# B&R Automation Studio project pneutrunk_plc_interface
Automation Studio 4.9

## Configuration Config1

### Task classes (Cpu.sw)
```
Cyclic#1:
  Client <- Source.UDP.Client.prg
  Narazy <- Source.Narazy.prg [disabled]
  Server <- Source.UDP.Server.prg
  Receiver <- (binary)
  Sender <- (binary)
Cyclic#4:
  Receiver1 <- Source.RS485.Receiver.prg
  Sender1 <- Source.RS485.Sender.prg
  Sensors <- Source.Sensors.prg
DataObjects: Acp10sys
Binaries: FWRules, TCData, udbdef, asfw, User, iomap, sysconf, arconfig, ashwd, Role, ashwac, Acp10map, acp10cfg
Libraries: runtime, AsUDP, asstring, standard, sys_lib, brsystem, dvframe, AsTCP, AsArLog, asieccon, astime, powerlnk, fileio
```

### IoMap.iom - X20CP1684/IoMap.iom
```iecst
VAR_CONFIG
	::modul.tlak2[5] AT %QW."X20CM8281".AnalogOutput01;
	::modul.tlak3[5] AT %QW."X20CM8281a".AnalogOutput01;
	::modul.tlak1[0] AT %QW."X20AO4622".AnalogOutput01;
	::modul.tlak2[0] AT %QW."X20AO4622".AnalogOutput02;
	::modul.tlak3[0] AT %QW."X20AO4622".AnalogOutput03;
	::modul.tlak1[1] AT %QW."X20AO4622".AnalogOutput04;
	::modul.tlak2[1] AT %QW."X20AO4622a".AnalogOutput01;
	::modul.tlak3[1] AT %QW."X20AO4622a".AnalogOutput02;
	::modul.tlak1[2] AT %QW."X20AO4622a".AnalogOutput03;
	::modul.tlak2[2] AT %QW."X20AO4622a".AnalogOutput04;
	::modul.tlak3[2] AT %QW."X20AO4622b".AnalogOutput01;
	::modul.tlak1[3] AT %QW."X20AO4622b".AnalogOutput02;
	::modul.tlak2[3] AT %QW."X20AO4622b".AnalogOutput03;
	::modul.tlak3[3] AT %QW."X20AO4622b".AnalogOutput04;
	::modul.tlak1[4] AT %QW."X20AO4622c".AnalogOutput01;
	::modul.tlak2[4] AT %QW."X20AO4622c".AnalogOutput02;
	::modul.tlak3[4] AT %QW."X20AO4622c".AnalogOutput03;
	::modul.tlak1[5] AT %QW."X20AO4622c".AnalogOutput04;
	::modul.tlakLinear AT %QW."X20CM8281b".AnalogOutput01;
	::modul.tlak2[6] AT %QW."X20AO4622d".AnalogOutput01;
	::modul.tlak3[6] AT %QW."X20AO4622d".AnalogOutput02;
	::modul.tlak1[6] AT %QW."X20AO4622d".AnalogOutput03;
	::buttons.stropCervenaLED AT %QX."X20DO9322".DigitalOutput08;
	::buttons.startLED AT %QX."X20DO9322".DigitalOutput06;
	::buttons.stopLED AT %QX."X20DO9322".DigitalOutput07;
	::buttons.stropBielaLED AT %QX."X20DO9322".DigitalOutput05;
	::buttons.startButton AT %IX."X20DM9324".DigitalInput01;
	::buttons.stop AT %IX."X20DM9324".DigitalInput02;
	::buttons.centralStop AT %IX."X20DM9324".DigitalInput04;
	::buttons.klucik AT %IX."X20DM9324".DigitalInput03;
END_VAR
```

## Logical view

### Global.typ
```iecst
TYPE
	tlacidla : 	STRUCT
		start : BOOL;
		ros : BOOL;
		stopLED : BOOL;
		stop : BOOL;
		startLED : BOOL;
		startButton : BOOL;
		centralStop : BOOL;
		stropBielaLED : BOOL;
		stropCervenaLED : BOOL;
		klucik : BOOL;
	END_STRUCT;
	automatic : 	STRUCT
		y_desired : ARRAY[0..6]OF REAL := [7(0.0)];
		x_desired : ARRAY[0..6]OF REAL := [7(0.0)];
		linear : INT;
		ball_up : BOOL;
		casovac : BOOL;
		effector : BOOL;
		casovac_uchopenie : BOOL;
		ball_piston : BOOL;
		novyCyklus : TIME := T#1s;
		novyCyklusStart : BOOL;
		trajectoryStart2 : BOOL;
		trajectoryTime2 : TIME := T#6s;
		automatic : BOOL;
		holdPosition : BOOL;
		cas : INT;
		box : INT;
		step_color : INT;
		popcorn : BOOL;
		testFarba : INT;
		loptickyVzasobniku : BOOL := TRUE;
		x_desired_previous : ARRAY[0..6]OF INT;
		y_desired_previous : ARRAY[0..6]OF INT;
		I_konstanta : ARRAY[0..6]OF INT;
		levitacia : BOOL;
		desiredPressure2 : ARRAY[0..6]OF INT;
		desiredPressure3 : ARRAY[0..6]OF INT;
		desiredPressure3_previous : ARRAY[0..6]OF INT;
		desiredPressure2_previous : ARRAY[0..6]OF INT;
		desiredPressure1_previous : ARRAY[0..6]OF INT;
		desiredPressureLinear : INT;
		desiredPressure1 : ARRAY[0..6]OF INT;
		step_repeatability : INT;
		handControl : BOOL;
		experiment2 : BOOL;
		experiment3 : BOOL;
		experiment1 : BOOL;
	END_STRUCT;
	packetRS485 : 	STRUCT
		packet : ARRAY[0..9]OF BYTE;
		sendPacketLED : ARRAY[0..5]OF BYTE;
		sendPacketSnimace : ARRAY[0..5]OF BYTE;
		sendPacketFinal : ARRAY[0..5]OF BYTE;
		id : USINT;
	END_STRUCT;
	packetUDP : 	STRUCT
		qLength : INT;
		c : INT;
		q : INT;
		qFull : STRING[80];
		comma : INT;
		qString : ARRAY[0..14]OF STRING[6];
		qDesired : ARRAY[0..14]OF REAL;
		color : INT;
		step : INT;
	END_STRUCT;
	tlaky : 	STRUCT
		tlak3 : USINT;
		tlak2 : USINT;
		tlak1 : USINT;
	END_STRUCT;
	moduly : 	STRUCT
		uhol2 : ARRAY[0..6]OF REAL := [7(0.0)];
		uhol1 : ARRAY[0..6]OF REAL := [7(0.0)];
		koncak : ARRAY[0..6]OF BOOL;
		led : ARRAY[0..6]OF BOOL;
		uholINT2 : INT;
		uholINT1 : INT;
		tlak1 : ARRAY[0..6]OF INT;
		tlak2 : ARRAY[0..6]OF INT;
		tlak3 : ARRAY[0..6]OF INT;
		tlakLinear : INT;
		alpha : ARRAY[0..6]OF REAL; (*uhol ktory posiela PLC do PC po odpocitani odchylky naklonenia realneho robota*)
		beta : ARRAY[0..6]OF REAL; (*uhol ktory posiela PLC do PC po odpocitani odchylky naklonenia realneho robota*)
		linearReal : REAL;
		naraz : ARRAY[0..7]OF BOOL;
		narazAktivny : BOOL;
	END_STRUCT;
END_TYPE
```

### Global.var
```iecst
VAR
	packetPos : packetUDP;
	packet485 : packetRS485;
	modul : moduly;
	buttons : tlacidla;
END_VAR
```

### Program Logical/Source/Sensors

#### Cyclic.st
```iecst
PROGRAM _CYCLIC

	modul.alpha[0]:= modul.uhol1[0]*1.0233 + 88.745;
	modul.alpha[1]:= modul.uhol1[1]*1.0228 + 88.871;
	modul.alpha[2]:= modul.uhol1[2]*1.0235 + 90.761;
	modul.alpha[3]:= modul.uhol1[3]*1.0254 + 88.307;
	modul.alpha[4]:= modul.uhol1[4]*1.0216 + 90.3;
	modul.alpha[5]:= modul.uhol1[5]*1.0039 + 87.274;
	modul.alpha[6]:= modul.uhol1[6]*1.0065 + 87.623;

	modul.beta[0]:= modul.uhol2[0]*1.0275 + 89.292;
	modul.beta[1]:= modul.uhol2[1]*1.0079 + 89.873;
	modul.beta[2]:= modul.uhol2[2]*1.043 + 92.476;
	modul.beta[3]:= modul.uhol2[3]*1.0308 + 90.739;
	modul.beta[4]:= modul.uhol2[4]*1.008 + 86.877;
	modul.beta[5]:= modul.uhol2[5]*1.0009 + 87.856;
	modul.beta[6]:= modul.uhol2[6]*1.0258 + 90.567;

END_PROGRAM
```

### LibAsUDP1_ST.typ
```iecst
(********************************************************************
 * COPYRIGHT -- Bernecker + Rainer
 ********************************************************************
 * File: Global.typ
 * Author: Bernecker + Rainer
 * Created: June 02, 2008
 ********************************************************************
 * Global data types of project LibAsUDP
 ********************************************************************)

TYPE
	LibAsUDP1_ST_typ : 	STRUCT  (*Datatyp for global Variables*)
		receive_data : ARRAY[0..100]OF UDINT; (*Data which has been received*)
		send_data : STRING[80]; (*Data which should be sent*)
	END_STRUCT;
END_TYPE
```

### Program Logical/Source/UDP/Client

#### Client.st
```iecst
(********************************************************************
 * COPYRIGHT -- Bernecker + Rainer
 ********************************************************************
 * Program: Client
 * File: Client.st
 * Author: Bernecker + Rainer
 * Created: June 02, 2008
 ********************************************************************
 * Implementation of program Client
 ********************************************************************)

PROGRAM _CYCLIC

	// 7/3/2025

	memset(ADR(LibAsUDP1_ST.send_data), 0, SIZEOF(LibAsUDP1_ST.send_data));
	memset(ADR(helpString), 0, SIZEOF(helpString));

	FOR i:=0 TO 6 BY 1 DO
		ftoa(modul.alpha[i], ADR(helpString));
		strcat(ADR(LibAsUDP1_ST.send_data), ADR(helpString));
		strcat(ADR(LibAsUDP1_ST.send_data), ADR(','));
		ftoa(modul.beta[i], ADR(helpString));
		strcat(ADR(LibAsUDP1_ST.send_data), ADR(helpString));
		strcat(ADR(LibAsUDP1_ST.send_data), ADR(','));
	END_FOR

	//LibAsUDP1_ST.send_data[0] := LibAsUDP1_ST.send_data[0] + 1;  (* Generate a "running" variable for Data transfer *)
	//LibAsUDP1_ST.send_data := '20.12 12.54 10.24 -13.25';

	(*
	memset(ADR(LibAsUDP1_ST.send_data), 0, SIZEOF(LibAsUDP1_ST.send_data));
	memset(ADR(helpString), 0, SIZEOF(helpString));

	FOR i:=0 TO 6 BY 1 DO
		ftoa(modul.uhol_XminusRef[i], ADR(helpString));
		strcat(ADR(LibAsUDP1_ST.send_data), ADR(helpString));
		strcat(ADR(LibAsUDP1_ST.send_data), ADR(','));
		ftoa(modul.uhol_YminusRef[i], ADR(helpString));
		strcat(ADR(LibAsUDP1_ST.send_data), ADR(helpString));
		strcat(ADR(LibAsUDP1_ST.send_data), ADR(','));
	END_FOR
	ftoa(modul.linearReal, ADR(helpString)); // vymenit za linearny
	strcat(ADR(LibAsUDP1_ST.send_data), ADR(helpString));
	*)
	//strcat(ADR(LibAsUDP1_ST.send_data), ADR(','));

	(*
	memset(ADR(LibAsUDP1_ST.send_data), 0, SIZEOF(LibAsUDP1_ST.send_data));
	memset(ADR(helpString), 0, SIZEOF(helpString));

	FOR i:=0 TO 5 BY 1 DO
		ftoa(modul.uhol1[i], ADR(helpString));
		strcat(ADR(LibAsUDP1_ST.send_data), ADR(helpString));
		strcat(ADR(LibAsUDP1_ST.send_data), ADR(','));
		ftoa(modul.uhol2[i], ADR(helpString));
		strcat(ADR(LibAsUDP1_ST.send_data), ADR(helpString));
		strcat(ADR(LibAsUDP1_ST.send_data), ADR(','));
	END_FOR
	ftoa(modul.uhol2[0], ADR(helpString)); // vymenit za linearny
	strcat(ADR(LibAsUDP1_ST.send_data), ADR(helpString));
	//strcat(ADR(LibAsUDP1_ST.send_data), ADR(','));
	*)
	CASE Client.sStep OF

		0:	(* Open UDP Port *)
			Client.UdpOpen_0.enable := 1;
			Client.UdpOpen_0.pIfAddr := 0;	(* Listen on all TCP/IP Interfaces*)
			Client.UdpOpen_0.port := 12051;	(* Port to listen*)
			Client.UdpOpen_0.options := 0;
			Client.UdpOpen_0;	(* Call the Function*)

			IF Client.UdpOpen_0.status = 0 THEN  (* UdpOpen successful*)
				Client.sStep := 1;
			ELSIF Client.UdpOpen_0.status = ERR_FUB_BUSY THEN  (* UdpOpen not finished -> redo *)
			  (* Busy *)
			ELSE  (* Goto Error Step *)
				Client.sStep := 10;
			END_IF

		1:	(* Send Data to the Server *)
			Client.server_address := '192.168.1.47';	(* IP Address of the Server *)
			Client.server_portnumber := 12050;	(* Port number of the Server *)

			Client.UdpSend_0.enable := 1;
			Client.UdpSend_0.ident := Client.UdpOpen_0.ident;	(* Connection Ident from AsUDP.UDP_Open *)
			Client.UdpSend_0.pHost := ADR(Client.server_address);
			Client.UdpSend_0.port := Client.server_portnumber;
			Client.UdpSend_0.pData := ADR(LibAsUDP1_ST.send_data);	(* Which data to send *)
			Client.UdpSend_0.datalen := SIZEOF(LibAsUDP1_ST.send_data);	(* Lenght of data to send *)
			Client.UdpSend_0.flags := 0;
			Client.UdpSend_0;	(* Call the Function*)

			IF Client.UdpSend_0.status = 0 THEN  (* Data sent *)
				Client.sStep := 2;
			ELSIF Client.UdpSend_0.status = ERR_FUB_BUSY THEN  (* UdpSend not finished -> redo *)
			  (* Busy *)
			ELSE  (* Goto Error Step *)
				Client.sStep := 10;
			END_IF

		2:	(* Receive Data from the Server *)
			Client.UdpRecv_0.enable := 1;
			Client.UdpRecv_0.ident := Client.UdpOpen_0.ident;  (* Connection Ident from AsUDP.UDP_Open *)
			Client.UdpRecv_0.pData	:= ADR(LibAsUDP1_ST.receive_data);  (* Where to store the incoming data *)//ADR(LibAsUDP1_ST.receive_data);
			Client.UdpRecv_0.datamax := SIZEOF(LibAsUDP1_ST.receive_data);  (* Lenght of data buffer *)
			Client.UdpRecv_0.flags := 0;
			Client.UdpRecv_0;  (* Call the Function*)

			IF Client.UdpRecv_0.status = 0 THEN  (* Data was received successfully -> Send next packet *)
				Client.sStep := 3;
				Client.no_data_received_count := 0;
			ELSIF Client.UdpRecv_0.status = udpERR_NO_DATA THEN  (* No data received - wait *)
			  (* No Data received *)
			  	Client.no_data_received_count := Client.no_data_received_count + 1;	(* Increase if no data are received *)

				IF Client.no_data_received_count > 200 THEN		(* No data timeout for TC1 [10ms] *)
					Client.no_data_received_count := 0;
					Client.sStep := 1;	(* Send again *)
				END_IF
			ELSIF Client.UdpRecv_0.status = ERR_FUB_BUSY THEN  (* UdpRecv not finished -> redo *)
			  (* Busy *)
			ELSE  (* Goto Error Step *)
				Client.sStep := 10;
			END_IF

		3: (* Close connection *)
			Client.UdpClose_0.enable := 1;
			Client.UdpClose_0.ident := Client.UdpOpen_0.ident;  (* Connection Ident from AsUDP.UDP_Open *)
			Client.UdpClose_0;  (* Call the Function*)

			IF Client.UdpClose_0.status = 0 THEN  (* Close successful -> Reopen the interface *)
				Client.sStep := 0;
			ELSIF Client.UdpClose_0.status = ERR_FUB_BUSY THEN  (* UdpClose not finished -> redo *)
			  (* Busy *)
			ELSE  (* Goto Error Step *)
				Client.sStep := 10;
			END_IF

		10: (* Here some error Handling has to be implemented *)

	END_CASE

END_PROGRAM
```

### Program Logical/Source/UDP/Server

#### Server.st
```iecst
(********************************************************************
 * COPYRIGHT -- Bernecker + Rainer
 ********************************************************************
 * Program: Server
 * File: Server.st
 * Author: Bernecker + Rainer
 * Created: June 02, 2008
 ********************************************************************
 * Implementation of program Server
 ********************************************************************)

PROGRAM _CYCLIC

	CASE Server.sStep OF

		0:	(* Open UDP Port *)
			Server.UdpOpen_0.enable := 1;
			Server.UdpOpen_0.pIfAddr := 0;	(* Listen on all TCP/IP Interfaces*)
			Server.UdpOpen_0.port := 12050;	(* Port to listen*)
			Server.UdpOpen_0.options := 0;
			Server.UdpOpen_0;	(* Call the Function*)

			IF Server.UdpOpen_0.status = 0 THEN  (* UdpOpen successful*)
				Server.sStep := 1;
			ELSIF Server.UdpOpen_0.status = ERR_FUB_BUSY THEN  (* UdpOpen not finished -> redo *)
			  (* Busy *)
			ELSE  (* Goto Error Step *)
				Server.sStep := 10;
			END_IF

		1:	(* Wait for Data *)
			Server.UdpRecv_0.enable := 1;
			Server.UdpRecv_0.ident := Server.UdpOpen_0.ident;	(* Client Ident from AsUDP.UDP_Open *)
			Server.UdpRecv_0.pData := ADR(Server.data_buffer);	(* Where to store the incoming data *)
			Server.UdpRecv_0.datamax := SIZEOF(Server.data_buffer);	(* Lenght of data buffer *)
			Server.UdpRecv_0.flags := 0;
			Server.UdpRecv_0.pIpAddr := ADR(Server.client_address);	(* IP Address of the Client *)
			Server.UdpRecv_0;	(* Call the Function*)

			IF Server.UdpRecv_0.status = 0 THEN  (* Data received *)
				Server.sStep := 2;
			ELSIF Server.UdpRecv_0.status = udpERR_NO_DATA THEN  (* No data received - wait *)
			  (* No Data received *)
			ELSIF Server.UdpRecv_0.status = ERR_FUB_BUSY THEN  (* UdpRecv not finished -> redo *)
			  (* Busy *)
			ELSE  (* Goto Error Step *)
				Server.sStep := 10;
			END_IF

		2:	(* Send Data back to Client *)

			Server.UdpSend_0.enable := 1;
			Server.UdpSend_0.ident := Server.UdpOpen_0.ident;	// Client Ident from AsUDP.UDP_Open
			Server.UdpSend_0.pHost := ADR(Server.client_address);	// IP Address of the Client
			Server.UdpSend_0.port := Server.UdpRecv_0.port;		// Port number of the Client
			Server.UdpSend_0.pData := ADR(Server.data_buffer);	// Which data to send
			Server.UdpSend_0.datalen := SIZEOF(Server.data_buffer);	// Lenght of data to send
			Server.UdpSend_0.flags := 0;
			Server.UdpSend_0;	// Call the Function

			(*
			Server.UdpSend_0.enable := 1;
			Server.UdpSend_0.ident := Server.UdpOpen_0.ident;	// Client Ident from AsUDP.UDP_Open
			Server.UdpSend_0.pHost := ADR(Server.client_address);	// IP Address of the Client
			Server.UdpSend_0.port := Server.UdpRecv_0.port;		// Port number of the Client
			Server.UdpSend_0.pData := ADR(Server.data_buffer);	// Which data to send
			Server.UdpSend_0.datalen := SIZEOF(Server.data_buffer);	// Lenght of data to send
			Server.UdpSend_0.flags := 0;
			Server.UdpSend_0;	// Call the Function

			packetPos.q := FIND(Server.data_buffer, 'q:');
			packetPos.c := FIND(Server.data_buffer, 'c:'); // Server.data_buffer bolo povodne ked to slo STRING[5][0..100] a tu bolo Server.data_buffer[0]
			packetPos.qLength := UDINT_TO_INT(Server.UdpSend_0.datalen) - (packetPos.q + 1) - packetPos.c;
			packetPos.qFull := MID(Server.data_buffer, packetPos.c-packetPos.q-2, packetPos.q+2);
			FOR i:=0 TO 13 BY 1 DO	//11
				packetPos.comma := FIND(packetPos.qFull, ',');
				packetPos.qString[i] := MID(packetPos.qFull, packetPos.comma, 0);
				packetPos.qFull := DELETE(packetPos.qFull, packetPos.comma+1, 0);
				packetPos.qDesired[i] := atof(ADR(packetPos.qString[i])) ;
			END_FOR
			packetPos.qString[14] := MID(packetPos.qFull, packetPos.comma, 0);//12
			packetPos.qFull := DELETE(packetPos.qFull, packetPos.comma+1, 0);
			packetPos.qDesired[14] := atof(ADR(packetPos.qString[14]));//12
			*)

			IF Server.UdpSend_0.status = 0 THEN  (* Data sent *)
				Server.sStep := 1;
			ELSIF Server.UdpSend_0.status = ERR_FUB_BUSY THEN  (* UdpSend not finished -> redo *)
			  (* Busy *)
			ELSE  (* Goto Error Step *)
				Server.sStep := 10;
			END_IF

		10:  (* Here some error Handling has to be implemented *)

	END_CASE

END_PROGRAM
```
